Fanuc KAREL source: kb00121.KL

-- PROVISIONAL review KL for V940-1; original PC SHA256 f25365e6f1cb9faf5fce8dc801889e774373734256ff5fa1a68f9b2d4001682b
-- Incomplete behavior may be omitted. Consult companion uncertainty JSON. Do not deploy.
PROGRAM KB00121
%NOLOCKGROUP
BEGIN
  -- V9_ZERO_TABLE_METADATA_HINT layout=0002_ascii; no indexed target words; source/name/runtime held
  -- UNRESOLVED_PC offsets 5-12; opcodes 9D,23
  -- UNRESOLVED_PC offsets 17-24; opcodes 9D,23
  -- UNRESOLVED_PC offsets 29-39; opcodes 9D,22,9D,33,35
  -- UNRESOLVED_PC offsets 44-51; opcodes 9D,23
  -- UNRESOLVED_PC offsets 56-90; opcodes 27,22,22,22,22,22,31
  -- UNRESOLVED_PC offsets 95-99; opcodes 7F
END KB00121
